# EPICS alarm handler configuration: mps_database/bareTest/alarms/areas/mpln_spd_mp01.alhConfig
GROUP NULL MPLN:SPD:MP01:1
$ALIAS MPS Link Node 92
$GUIDANCE
LTUH MPS
   Group Name: MPLN:SPD:MP01:1
   Summary PV:  MPLN:SPD:MP01:1:STATSUMY
$END
CHANNEL  MPLN:SPD:MP01:1    MPLN:SPD:MP01:1:MPS_EN_RBV		-----
CHANNEL  MPLN:SPD:MP01:1    MPLN:SPD:MP01:1:LC1_MODE_RBV		-----
